{attribute 'TcGenerated'}
{attribute 'no-analysis'}
{attribute 'linkalways'}
// This function has been automatically generated from the project information.
VAR_GLOBAL CONSTANT
    {attribute 'const_non_replaced'}
    stLibVersion_LCLSVacuumSerialDriverLib : ST_LibVersion := (iMajor := 1, iMinor := 3, iBuild := 2, iRevision := 0, nFlags := 1, sVersion := '1.3.2');
END_VAR

(* stored: Version 1.1.0.1, ProductVersion 3.1.4018.5
   GVL Global_Version: Id {f757f888-2bdd-462c-ba79-93f7505eedaa} *)
